Yaskawa INFORM job: R1_W43-44-A3(0,180)_MOD.JBI

/JOB
//NAME R1_W43-44-A3(0,180)_MOD
///FOLDERNAME KRIS-SCIANA
//POS
///NPOS 44,44,0,5,0,0
///TOOL 0
///POSTYPE PULSE
///PULSE
C00000=100690,117515,19281,-12198,92695,84321
C00001=120646,105623,43243,-26574,112528,70688
C00002=121274,154245,111368,-24314,97313,74325
C00003=121274,154438,114214,-24210,95800,74637
C00004=121274,154851,115862,-24167,95064,74788
C00005=121274,154780,115625,-24172,95164,74767
C00006=121276,146733,104349,-24344,97732,74240
C00007=121558,133388,85971,-25011,99218,71019
C00008=122962,94279,37460,-27911,94090,53096
C00009=122329,94216,37382,-27741,93916,52921
C00010=123209,97456,36086,-28128,96366,52631
C00011=120383,157389,107739,-24594,100575,73316
C00012=116229,162405,111560,-14744,100873,1862
C00013=115459,106900,46533,30387,111082,-71354
C00014=114147,129060,50437,24217,120657,-71531
C00015=111807,128387,53992,23721,118891,-72790
C00016=111807,127177,53688,23616,118490,-72883
C00017=111807,127341,53728,23631,118546,-72870
C00018=111737,124719,50040,23867,119410,-72694
C00019=111793,127538,53115,23751,118989,-72773
C00020=105106,126619,61759,43830,113933,-71432
C00021=105742,125955,60839,43837,113819,-71196
C00022=105247,126467,61549,43833,113909,-71377
C00023=104625,101741,30044,44640,106766,-73909
C00024=105775,127046,63338,43498,113088,-71528
C00025=105564,121676,55912,44152,114511,-70943
C00026=104923,123258,56815,44322,114981,-71008
C00027=109200,142517,76554,28006,119167,-71726
C00028=109011,139908,74162,28039,119340,-71751
C00029=111572,137830,71231,28319,119221,-70759
C00030=111732,137715,71077,28333,119205,-70700
C00031=111445,141432,74405,28286,119171,-70824
C00032=110736,115247,37574,31685,127424,-68467
C00033=120646,105623,43243,-26574,112528,70688
C00034=125596,166598,109272,-39285,104070,72245
C00035=127750,114688,46201,-46149,96552,74998
C00036=124981,161828,106073,-39148,103426,72229
C00037=125023,138902,76078,-39156,109193,70185
C00038=125119,81574,11326,-35040,120442,67336
C00039=124901,86805,20326,-35271,122089,67752
C00040=122018,86472,19904,-35027,121163,66907
C00041=126050,83344,21642,-44995,117967,66728
C00042=126878,85259,21962,-45424,118894,66634
C00043=126878,84917,22081,-45314,118716,66728
BC00000=32768,605746,1075157
BC00001=176,523582,733596
BC00002=176,523582,733596
BC00003=176,523582,733596
BC00004=176,523582,733596
BC00005=176,523582,733596
BC00006=176,523582,733596
BC00007=176,523582,733596
BC00008=176,523582,733596
BC00009=176,523582,733596
BC00010=176,523582,733596
BC00011=176,564332,733596
BC00012=178188,564332,733596
BC00013=398029,538415,833874
BC00014=395342,503532,593108
BC00015=395342,503532,593108
BC00016=395342,503532,593108
BC00017=395342,503532,593108
BC00018=395342,503532,593108
BC00019=395342,503532,593108
BC00020=395342,503532,593108
BC00021=395342,503532,593108
BC00022=395342,503532,593108
BC00023=395342,503533,593107
BC00024=395342,503533,593107
BC00025=395342,503533,593107
BC00026=395342,503533,593107
BC00027=395342,503533,593107
BC00028=395342,503533,593107
BC00029=395342,503533,593107
BC00030=395342,503533,593107
BC00031=395342,503533,593107
BC00032=395342,545913,642597
BC00033=176,523582,733596
BC00034=31,523584,561235
BC00035=31,523584,561235
BC00036=31,523584,561235
BC00037=31,514484,583389
BC00038=31,469507,692894
BC00039=31,469507,692894
BC00040=32,469508,692894
BC00041=32,469508,692894
BC00042=32,469508,692894
BC00043=32,505316,714307
///POSTYPE BASE
///RECTAN
///RCONF 0,0,0,0,1,0,0,0,0,0,0,0,0,0,0,0,0,0,0,0,0,0,0,0
P00006=2.006,1.622,-0.565,0.0000,0.0000,0.0000
P00021=0.073,2.058,-0.109,0.0000,0.0000,0.0000
P00022=2.006,1.622,-0.565,0.0000,0.0000,0.0000
///RCONF 0,0,0,0,0,0,0,0,0,0,0,0,0,0,0,0,0,0,0,0,0,0,0,0
P00023=-2.957,-4.083,2.762,0.0000,0.0000,0.0000
P00024=-1.466,-0.226,-0.419,0.0000,0.0000,0.0000
//INST
///DATE 2025/05/08 14:38
///ATTR SC,RW
///GROUP1 RB1,BS1
NOP
SFTOF
MOVJ C00000 BC00000 VJ=100.00
MOVJ C00001 BC00001 VJ=100.00
MOVL C00002 BC00002 V=83.3
MOVL C00003 BC00003 V=83.3
REFP 3 C00004 BC00004
CALL JOB:SEARCH-R1
SET P021 P006
SFTON P021
MOVL C00005 BC00005 V=83.3
REFP 3 C00006 BC00006
CALL JOB:SEARCH-R1
SET P021 P006
SFTON P021
MOVL C00007 BC00007 V=83.3
MOVL C00008 BC00008 V=83.3
REFP 3 C00009 BC00009
CALL JOB:SEARCH-R1
SET P022 P006
SFTON P022
MOVL C00010 BC00010 V=83.3
SFTOF
MOVJ C00011 BC00011 VJ=100.00
MOVJ C00012 BC00012 VJ=100.00
MOVJ C00013 BC00013 VJ=100.00
MOVL C00014 BC00014 V=166.7
MOVL C00015 BC00015 V=83.3
REFP 3 C00016 BC00016
CALL JOB:SEARCH-R1
SET P023 P006
SFTON P023
MOVL C00017 BC00017 V=83.3
REFP 3 C00018 BC00018
CALL JOB:SEARCH-R1
SET P023 P006
SFTON P023
MOVL C00019 BC00019 V=83.3
MOVL C00020 BC00020 V=83.3
REFP 3 C00021 BC00021
CALL JOB:SEARCH-R1
SET P024 P006
SFTON P024
MOVL C00022 BC00022 V=83.3
MACRO1 MJ#(0) ARGF6
MOVL C00023 BC00023 V=83.3 PL=0
ARCON
MOVL C00024 BC00024 V=8.3
MOVL C00025 BC00025 V=8.3
ARCOF
MOVL C00026 BC00026 V=83.3
SFTON P023
MOVL C00027 BC00027 V=83.3
MOVL C00028 BC00028 V=83.3 PL=0
ARCON
MOVL C00029 BC00029 V=10.8
SFTON P024
MOVL C00030 BC00030 V=10.8
ARCOF
MOVL C00031 BC00031 V=83.3
SFTOF
MOVJ C00032 BC00032 VJ=100.00
MOVJ C00033 BC00033 VJ=100.00
SFTON P022
MOVL C00034 BC00034 V=83.3
MACRO1 MJ#(0) ARGF6
MOVL C00035 BC00035 V=83.3 PL=0
ARCON
MOVL C00036 BC00036 V=8.3
ARCOF
MOVL C00037 BC00037 V=83.3
SFTON P021
MOVL C00038 BC00038 V=83.3
MOVL C00039 BC00039 V=83.3 PL=0
ARCON
MOVL C00040 BC00040 V=10.8
SFTON P022
MOVL C00041 BC00041 V=10.8
ARCOF
MOVL C00042 BC00042 V=83.3
SFTOF
MOVJ C00043 BC00043 VJ=100.00
END
